(* IEC 61131-3 sources: InfiniteStateMachine/st/project/infinitestatemachine/interfaces/istate, 2 files *)

(* ---- enter-Enter.st ---- *)
(* --- Interface --- *)
METHOD Enter
VAR_INPUT
	fbStateMachine : StateMachine;
END_VAR

(* ---- leave-Leave.st ---- *)
(* --- Interface --- *)
METHOD Leave
VAR_INPUT
	fbStateMachine : StateMachine;
END_VAR
